// TIA Portal V19 export
DATA_BLOCK "DI WATER TRANSFER DB"   // DB170
{ S7_Optimized_Access := 'TRUE' }
// stored: MemoryReserve 100
   VAR
      "P-502 AB/BC/CA" : Bool;
   END_VAR
BEGIN
END_DATA_BLOCK
